FUNCTION FC_BYTE_TO_BOOLARR
VAR_INPUT
	pMyBool : POINTER TO BOOL; // Destination 
	pMyByte : POINTER TO BYTE; // Source   
	nSize	: UINT;               
END_VAR
VAR
    i : UINT;                       
	myBools : ARRAY[0..7] OF BOOL; 
END_VAR

FOR i:= 0 TO nSize-1 BY 8 DO
	myBools := FC_BYTE_TO_BOOLBYTE(pMyByte[i/8]);
	MEMCPY(ADR(pMyBool[i]), ADR(myBools), SIZEOF(myBools));
END_FOR

END_FUNCTION

(* stored: Version 1.1.0.1, ProductVersion 3.1.4024.13
   POU FC_BYTE_TO_BOOLARR: Id {ff58ad71-d4a6-4014-afdb-be890f252e26}, SpecialFunc None *)
